{attribute 'qualified_only'}
VAR_GLOBAL
//	fbUpdateModue:FB_UPDATE_MODULE;
	
	fbDeviationCheck		:ARRAY[1..29] OF FB_DeviationCheck;
	fbSensorLimitCheck		:ARRAY[1..7] OF FB_SensorLimitCheck;  // Pressure N2 H2 H2S,H2SE + Reactor / Press / Roration
	fbFaultCheck			:ARRAY[1..8] OF FB_FaultCheck; // CDA/CoolingWafer/Rotation Fault/Vacuum Pump Fault/Gas Cabinet Open / Reactor Door Open / Dor Fault
END_VAR

(* stored: Version 1.1.0.1, ProductVersion 3.1.4024.12
   GVL GVL_SEQUENCE: Id {afa24cfe-a057-4c9d-bd84-b82c36777d71} *)
